FUNCTION_BLOCK fbUldConveyor3Zones
VAR_INPUT

	bEnable		: BOOL;
	bRapidPB	: BOOL;
	bUldBasketZone1TransferMemoryBit: BOOL;
	bUldBasketZone1ConfirmMemoryBit: BOOL;
	bUldBasketZone2TransferMemoryBit: BOOL;
	bUldBasketZone2ConfirmMemoryBit	: BOOL;

	bUldSensor1: BOOL;
	bUldSensor2: BOOL;
	bUldEndSensor: BOOL;
(*
	diZone1BasketConfirmDelayTime	: DINT;
	diZone2BasketConfirmDelayTime	: DINT;
	diRapidPBDelayTime	: DINT;
*)
	diEndZoneBasketConfirmDelayTime	: DINT;

	bEmergencyStop: BOOL;
END_VAR
VAR_OUTPUT
	bMotorOnOff	: BOOL;
END_VAR
VAR
	bRapidPBRE: R_TRIG;
	bMotorStopBit: BOOL;
	TON1: TON;
	TON2: TON;
	bConvAutoCut: BOOL;

	(*TRIG1: R_TRIG;
	Trig2: R_TRIG;
	TON3: TON;
	RampIn: BOOL;
	TON4: TON;
	CVDelayOff : BOOL;
	TON5: TON;*)

END_VAR

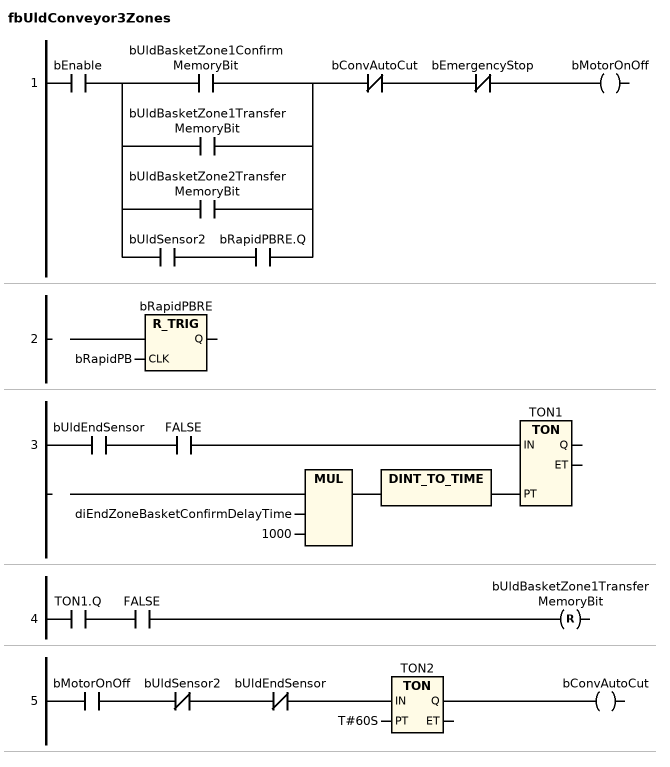
// NETWORK 1
bMotorOnOff := (bEnable AND (bUldBasketZone1ConfirmMemoryBit OR bUldBasketZone1TransferMemoryBit OR bUldBasketZone2TransferMemoryBit OR bUldSensor2 AND bRapidPBRE.Q)) AND NOT bConvAutoCut AND NOT bEmergencyStop;

// NETWORK 2
bRapidPBRE(CLK := bRapidPB); // R_TRIG

// NETWORK 3
TON1(IN := bUldEndSensor AND FALSE, PT := DINT_TO_TIME(diEndZoneBasketConfirmDelayTime * 1000)); // TON

// NETWORK 4
bUldBasketZone1TransferMemoryBit R= TON1.Q AND FALSE;

// NETWORK 5
TON2(IN := bMotorOnOff AND NOT bUldSensor2 AND NOT bUldEndSensor, PT := T#60S); // TON
bConvAutoCut := TON2.Q;

END_FUNCTION_BLOCK

(* stored: Version 1.1.0.1, ProductVersion 3.1.4024.12
   POU fbUldConveyor3Zones: Id {dc201380-d9be-43ac-ba78-2de94ca4cb8d}, SpecialFunc None *)
